(* CoDeSys 2.3 export: ST_WB_VALVE_LS_CFG.EXP *)

(* Data type *)
TYPE ST_WB_VALVE_LS_CFG :
STRUCT
	Cycle   : REAL; (*Seconds*)
	TimeMax : REAL; (*Seconds*)
	PushTime: REAL; (*Seconds*)
	PushP   : REAL; (*Bar*)

	TgtLS_Half : REAL;
	LS_DB   : REAL;

	HP      : BYTE; (*Num. Pumps*)
END_STRUCT
END_TYPE
